TYPE outWord :
STRUCT
	Lower : USINT; //Lower Bytes
	Upper : USINT; //Upper Bytes
END_STRUCT
END_TYPE

(* stored: Version 1.1.0.1, ProductVersion 3.1.4024.12
   DUT outWord: Id {782a6a73-ba1a-4328-b2c1-96a7aa705521} *)
